FUNCTION_BLOCK FB_PiezoDriveDS402PP EXTENDS FB_PiezoDriveDS402
VAR_INPUT
END_VAR
VAR_OUTPUT
END_VAR
VAR
    eDriveCmdState: E_DRIVE_CMD_STATE;
END_VAR

METHOD Brake : BOOL
SUPER^.Brake();
END_METHOD

METHOD DS402StateMachine
VAR_INPUT
END_VAR
SUPER^.DS402StateMachine();

IF SUPER^.DriveStateTransition = E_DriveStates.OPERATION_ENABLED THEN
    IF SUPER^.stPiezoStage.bMoveCmd THEN
        // call MoveAbsolute;
    END_IF
END_IF
END_METHOD

(*FB_Init is always available implicitly and it is used primarily for initialization.
The return value is not evaluated. For a specific influence, you can also declare the
methods explicitly and provide additional code there with the standard initialization
code. You can evaluate the return value.*)
METHOD FB_Init : BOOL
VAR_INPUT
    (* TRUE: the retain variables are initialized (reset warm / reset cold)*)
    bInitRetains	: BOOL;
    (* TRUE: the instance will be copied to the copy code afterward (online change)   *)
    bInCopyCode	: BOOL;
    stStage : REFERENCE TO ST_PiezoStage;
END_VAR
END_METHOD

METHOD Halt : BOOL
SUPER^.Halt();
END_METHOD

METHOD Home : BOOL
SUPER^.Home();
END_METHOD

METHOD Interlock : BOOL
SUPER^.Interlock();
END_METHOD

METHOD Logger : BOOL
SUPER^.Logger();
END_METHOD

METHOD MoveAbsolute

VAR
    checkVelocity : LREAL := 0.0;
    checkAcceleration : LREAL := 0.0;


END_VAR
SUPER^.MoveAbsolute();

IF SUPER^.AbsMoveEnabled THEN

    CASE eDriveCmdState OF
        E_DRIVE_CMD_STATE.PREPARE_MOTION_PARAMS:
        // Activate soft limit to avoid bumping hard on the end stops
        fMaxVelocity :=
        SUPER^.stPiezoStage.nTargetPosition := LREAL_TO_DINT (SUPER^.stPiezoStage.fPosition / MAX(SUPER^.stPiezoStage.fscalingFactor, 0.000000001));

        SUPER^.stPiezoStage.nProfilVelocity := LIMIT(1, LREAL_TO_DINT (SUPER^.stPiezoStage.fVelocity * MAX(SUPER^.stPiezoStage.fscalingFactor, 0.000000001), 1000);
        SUPER^.stPiezoStage.nProfilAcceleration := LREAL_TO_DINT (SUPER^.stPiezoStage.fAcceleration * MAX(SUPER^.stPiezoStage.fscalingFactor, 0.000000001));
        SUPER^.stPiezoStage.nProfilDecceleration := LREAL_TO_DINT (SUPER^.stPiezoStage.fAcceleration * MAX(SUPER^.stPiezoStage.fscalingFactor, 0.000000001));
        // this need to be handle in the power method and interlock to comfirm the move cmd
        // stPiezoStage.stAxisStatus.bExecute := stPiezoStage.bExecute;
        // stPiezoStage.stAxisStatus.nCommand := 10;

        stPiezoStage.nModeOfOperation := E_MODE_OF_OPERATION.PROFILE_POSITION;

        E_DRIVE_CMD_STATE.INITIATE_MOTION:;

        E_DRIVE_CMD_STATE.DRIVE_IN_MOTION:;
        E_DRIVE_CMD_STATE.TARGET_REACHED:
            // Prepare next move
            SUPER^.AbsMoveEnabled := FALSE;

    END_CASE
END_IF
END_METHOD

METHOD MoveVelocity : BOOL
END_METHOD

METHOD Power : BOOL
SUPER^.Power();
END_METHOD

METHOD Reset : BOOL
SUPER^.Reset();
END_METHOD

END_FUNCTION_BLOCK

(* stored: Version 1.1.0.1
   POU FB_PiezoDriveDS402PP: Id {6e47a4a9-16e3-49c8-8786-19fbbc700413}, SpecialFunc None
   Method Brake: Id {22a77937-1757-472e-8a24-02f41806a6fb}
   Method DS402StateMachine: Id {adad349e-6f22-41f6-bf4b-2c2ba773c644}
   Method FB_Init: Id {ea3b8a11-1b80-40a7-b145-7a2a5e25ca70}
   Method Halt: Id {a3eb5c8c-6142-41f2-a5f0-329f2aa7b09f}
   Method Home: Id {b3172138-e5cb-4d78-92a5-25024c9364c9}
   Method Interlock: Id {ace40c54-e822-492e-bd82-afe1a2bf1748}
   Method Logger: Id {f160a88a-3c4d-4691-a405-183a03bb632e}
   Method MoveAbsolute: Id {1452777d-f00c-4295-b378-678683e81128}
   Method MoveVelocity: Id {654fd94f-9d98-4616-85f0-4b450356f9ca}
   Method Power: Id {dd93fa86-0fa6-4325-a503-186f139a39d1}
   Method Reset: Id {0df62ddd-bca4-4bda-b598-c8f2f20db140} *)
